TYPE U_SAFETY_AND :
UNION
	stStatusWords					: ST_SAFETY_FBStatus;		(* BUnknown, BState, wDiagnosis, wInputs, wOutputs - takie same dla wszystkich FB *)
	stStatus						: ST_SAFETY_AND; 			(* Rozbite na Bity - inne dla kazdego bloku*)
END_UNION
END_TYPE

(* stored: Version 1.1.0.1, ProductVersion 3.1.4022.12
   DUT U_SAFETY_AND: Id {a159b007-2305-4343-ba9a-8ada1c98b11d} *)
